TYPE ASCF_State_Internals :
STRUCT
	Curr		: WORD		:= 16#0001;		//Current state of a state machine
	Prev		: WORD		:= 16#FFFF;		//Previous state of a state machine
END_STRUCT
END_TYPE

(* stored: Version 1.1.0.1, ProductVersion 3.1.4026.4
   DUT ASCF_State_Internals: Id {5d7b554e-6574-43d6-850a-bf760749dd99} *)
